(* CoDeSys 2.3 export: GLOBAL_VARIABLES.EXP *)

(* Global variable list: Global_Variables *)
VAR_GLOBAL CONSTANT
	_ERR_Nums: UINT := 5;
END_VAR

VAR_GLOBAL
	glbErrors: ARRAY [1.._ERR_Nums] OF _ERR :=
		(Msg := 'Активирована кнопка Аварийной остановки', Lock := TRUE, Zoomer := TRUE),
		(Msg := 'Активирована Пожарная Тревога', Latch := TRUE, Lock := TRUE, Zoomer := TRUE ),
		(Msg := 'Загрязнен возжушный фильтр', Zoomer := TRUE);




END_VAR
